{attribute 'linkalways'} 
{attribute 'no_explicit_call' := 'This FB is a CLASS and must be accessed using methods or properties'}
{attribute 'enable_dynamic_creation'}
FUNCTION_BLOCK Node_F_VN_CreateNDimensionalImageAndSetPixels EXTENDS VisionNode
VAR
    ipImage : _ITcVnImage;
    aShape : _TcVnArray33_UDINT;
    ePixelType : _ETcVnElementType(ETcVnElementType.TCVN_ET_USINT);
    fValue : _LREAL(0.0);
    hrPrev : _HRESULT(S_OK);
	hresult : _HRESULT(S_OK);
END_VAR

METHOD PUBLIC  Clone : I_Node
VAR
	pNode : POINTER TO Node_F_VN_CreateNDimensionalImageAndSetPixels;
END_VAR
pNode := __NEW(Node_F_VN_CreateNDimensionalImageAndSetPixels);
Clone := pNode^;
END_METHOD

METHOD FB_init : BOOL
VAR_INPUT
	bInitRetains : BOOL; // if TRUE, the retain variables are initialized (warm start / cold start)
	bInCopyCode : BOOL;  // if TRUE, the instance afterwards gets moved into the copy code (online change)
END_VAR
AddParameter('aShape', aShape);
AddParameter('ePixelType', ePixelType);
AddParameter('fValue', fValue);
AddInput('hrPrev', hrPrev);
AddOutput('ipImage', ipImage);
AddOutput('hresult',hresult);
END_METHOD

METHOD PROTECTED OnExecute
hresult.Value := F_VN_CreateNDimensionalImageAndSetPixels(
    ipImage := ipImage.Value,
    aShape := aShape.Value,
    ePixelType := ePixelType.Value,
    fValue := fValue.Value,
	hrPrev:= hrPrev.Value);
END_METHOD

METHOD PUBLIC PreExecutionCheck
VAR_INPUT
	Check : I_PreExecutionChecks;
END_VAR
END_METHOD

END_FUNCTION_BLOCK

(* stored: Version 1.1.0.1, ProductVersion 3.1.4024.13
   POU Node_F_VN_CreateNDimensionalImageAndSetPixels: Id {cf4b3bb3-1636-0d53-1eaa-78a25939a321}, SpecialFunc None
   Folder Constructor: Id {4df68378-0f35-0e8e-344c-85298fd73c6e}
   Method Clone: Id {6b5c5a5d-f0c0-0a78-261a-4b7c78b5eafe}
   Method FB_init: Id {a76ae431-a845-08f6-36ff-8fb0c5854e97}
   Method OnExecute: Id {93059fb3-38e9-06c9-30f3-bdeef426c10c}
   Method PreExecutionCheck: Id {e8799356-8ec8-06e6-0d84-b18bc2cb84bc} *)
